// TIA Portal V17 export
// export: Created 2022-06-18T11:46:49.493708Z, ExportSetting None, DisplayName Totally Integrated Automation Portal, DisplayVersion V17, DisplayName TIA Portal Openness, DisplayVersion V17, DisplayName TIA Portal Teamcenter Gateway, DisplayVersion V17, DisplayName TIA Portal Version Control Interface, DisplayVersion V17, DisplayName TIA Portal Test Suite Advanced, DisplayVersion V17, DisplayName SINAMICS Startdrive Advanced, DisplayVersion V17, DisplayName SINAMICS DCC, DisplayVersion V17, DisplayName SINAMICS Startdrive G130, G150, S120, S150, SINAMICS MV, S210, DisplayVersion V17, DisplayName SINAMICS Startdrive G110M, G120, G120C, G120D, G120P, G115D, DisplayVersion V17, DisplayName STEP 7 Professional, DisplayVersion V17, DisplayName SIMATIC Energy Suite, DisplayVersion V17, DisplayName STEP 7 CFC, DisplayVersion V17, DisplayName STEP 7 Safety, DisplayVersion V17, DisplayName WinCC Advanced / Unified PC, DisplayVersion V17, DisplayName SIMATIC Visualization Architect, DisplayVersion V17
DATA_BLOCK "InstanceDB_FB"   // DB7
// stored: InstanceOfName Lib_FB_Motor_DS_RotSens, InstanceOfType FB
"Lib_FB_Motor_DS_RotSens"
   // VAR_INPUT
   //    I_Initialization : Bool;
   //    IR_CycleTime : Real;
   //    II_Obj_ID : Int;
   //    I_CmdGeneralReset : Bool;
   //    I_One_1s : Bool;
   //    I_EnableHorn : Bool;
   //    I_EstopLocal : Bool;
   //    I_EstopHMI : Bool;
   //    I_SuppyBox_Ok : Bool;
   //    I_ELSS_On : Bool;
   //    I_MP_Ok : Bool;
   //    I_FeedbackForwardOn : Bool;
   //    I_FeedbackReverseOn : Bool;
   //    I_EnableForward : Bool;
   //    I_EnableReverse : Bool;
   //    I_Brake_Ok : Bool;
   //    I_Brake_CP_Ok : Bool;
   //    I_Cooling_FeedbackRun : Bool;
   //    I_Cooling_CP_Ok : Bool;
   //    I_GenFaultMainDrive : Bool;
   //    I_CmdAutoFromInputFB : Bool;
   //    I_CmdAutoForward : Bool;
   //    I_CmdAutoReverse : Bool;
   //    I_ManLocalModeActive : Bool;
   //    "I_CmdManLocalForward/Open" : Bool;
   //    "I_CmdManLocalReverse/Close" : Bool;
   //    IB_InterlocksForward_8 : Byte;
   //    IB_InterlocksReverse_8 : Byte;
   //    IW_ExternalError_16 : Word;
   //    I_ExternalWarning : Bool;
   //    I_RotationSensor : Bool;
   //    II_RotationSensorMode : Int;
   //    I_Termistor_Ok : Bool;
   //    IR_TimeTripKM : Real;
   //    IR_TimeTripCool : Real;
   //    IR_TimeTripBrake : Real;
   // END_VAR
   // VAR_OUTPUT
   //    Q_CmdForward : Bool;
   //    Q_CmdReverse : Bool;
   //    Q_CmdReleaseClutch : Bool;
   //    Q_CmdRunCooling : Bool;
   //    Q_CmdHorn : Bool;
   //    Q_Error : Bool;
   //    Q_Warning : Bool;
   //    Q_Auto : Bool;
   //    Q_ManLocal : Bool;
   //    Q_Stoped : Bool;
   //    Q_Run : Bool;
   //    Q_RunForward : Bool;
   //    Q_RunReverse : Bool;
   //    Q_DataErr : Bool;
   // END_VAR
   // VAR_IN_OUT
   //    IQ_PLC_CycleInfo : Variant;
   // END_VAR
   // VAR
   //    s_RequestForward : Bool;
   //    s_RequestReverse : Bool;
   //    s_Stopdown : Bool;
   //    s_StartCooling : Bool;
   //    s_ReleaseBrake : Bool;
   //    si_GenCountMotoHours : DInt;
   //    si_QuanStartsForward : DInt;
   //    si_QuanStartsReverse : DInt;
   //    s_EdgeAuto : "Lib_FB_Edge";
   //    s_EdgeSim : "Lib_FB_Edge";
   //    s_EdgeLocal : "Lib_FB_Edge";
   //    EdgeActivForward { ExternalAccessible := 'False'; ExternalVisible := 'False'; ExternalWritable := 'False'} : "Lib_FB_Edge";
   //    EdgeActivRevers { ExternalAccessible := 'False'; ExternalVisible := 'False'; ExternalWritable := 'False'} : "Lib_FB_Edge";
   // END_VAR
   // VAR RETAIN
   //    Simulation { ExternalAccessible := 'False'; ExternalVisible := 'False'; ExternalWritable := 'False'} : Struct
   //       Obj_DATA_BACKUP : Struct
   //          Config : "_Motor_DS_RotSens_Config";
   //          Counters : "_Motor_DS_RotSens_Counters";
   //          sud_MotoHours_Electro : "_MotoHours_One";
   //          sud_MotoHours_Mech : "_MotoHours_One";
   //       END_STRUCT;
   //    END_STRUCT;
   // END_VAR
   // VAR
   //    s_Moto : "Lib_FB_MotSimp";
   //    s_TON_TripBrake : "Lib_FB_Timer_ON_Simple";
   //    s_TON_TripCool : "Lib_FB_Timer_ON_Simple";
   //    s_TON_Horn : "Lib_FB_Timer_ON_Simple";
   //    s_fb_TurningSensor_Instance : "lib_fb_TurningSensor";
   // END_VAR
BEGIN
END_DATA_BLOCK
